Universal Robots PolyScope program: Calibration_6001.urp

Program Calibration_6001 (installation=GD directory=/programs/GD createdIn=5.13.0 lastSavedIn=5.13.0 robotSerialNumber=20205000017)
Calibrated DH parameters: a=[-0.000157, -0.56303, -0.236706, -0.000074, -0.000109, 0]; d=[0.181705, 47.632387, 369.599619, -417.058513, 0.119878, 0.115667]; alpha=[1.570881, -0.005074, -0.001247, 1.56886, -1.570997, 0]; deltaTheta=[0, -0.405485, 5.544791, 1.143886, -0.000009, -0.000001]
InitVariablesNode
BeforeStart
  Script file /programs/GD/ROVI/ROVI_RESET.script
    | def ROVI_RESET():
    |   if (not socket_open(host,port,socket_name)):
    |     rovi_err=902
    |     return False
    |   end
    |   socket_send_line("X0()",socket_name)
    |   ret=socket_read_line(socket_name,socket_timeout)
    |   if (ret == "OK"):
    |     rovi_err=0
    |   elif (ret == "NG"):
    |     rovi_err=to_num(socket_read_line(socket_name,socket_timeout))
    |   else:
    |     ret="NG"
    |     rovi_err=903
    |   end
    |   socket_close(socket_name)
    |   if (rovi_err != 0):
    |     if (is_popup):
    |       popup(str_cat(ret,rovi_err),title="X0",warning=True,blocking=True)
    |     end
    |     return False
    |   else:
    |     return True
    |   end
    | end
  Script file /programs/GD/ROVI/ROVI_CAPTURE.script
    | def ROVI_CAPTURE():
    | #  p=get_actual_tool_flange_pose()
    |   p=Bucket
    |   if (not socket_open(host,port,socket_name)):
    |     rovi_err=902
    |     return False
    |   end
    |   socket_send_string("X1(",socket_name)
    |   socket_send_string(p[0],socket_name)
    |   socket_send_string(",",socket_name)
    |   socket_send_string(p[1],socket_name)
    |   socket_send_string(",",socket_name)
    |   socket_send_string(p[2],socket_name)
    |   socket_send_string(",",socket_name)
    |   socket_send_string(p[3],socket_name)
    |   socket_send_string(",",socket_name)
    |   socket_send_string(p[4],socket_name)
    |   socket_send_string(",",socket_name)
    |   socket_send_string(p[5],socket_name)
    |   socket_send_line(")",socket_name)
    |   ret=socket_read_line(socket_name,socket_timeout)
    |   if (ret == "OK"):
    |     rovi_err=0
    |     f=socket_read_ascii_float(4,socket_name,socket_timeout)
    |     while (f[0]!=4):
    |       sleep(0.3)
    |       f=socket_read_ascii_float(4,socket_name,socket_timeout)
    |     end
    |     i=0
    |     while (i<4):
    |       Y1[i]=f[i+1]
    |       i=i+1
    |     end
    |   elif (ret == "NG"):
    |     rovi_err=to_num(socket_read_line(socket_name,socket_timeout))
    |   else:
    |     ret="NG"
    |     rovi_err=903
    |   end
    |   socket_close(socket_name)
    |   if (rovi_err != 0):
    |     if (is_popup):
    |       popup(str_cat(ret,rovi_err),title="X1",warning=True,blocking=True)
    |     end
    |     return False
    |   else:
    |     return True
    |   end
    | end
  Script file /programs/GD/ROVI/ROVI_SOLVE.script
    | def ROVI_SOLVE(is_popup=is_popup):
    |   buf=p[10000.0,0.0,0.0,0.0,0.0,0.0]
    |   if (not socket_open(host,port,socket_name)):
    |     rovi_err=902
    |     return False
    |   end
    |   socket_send_line("X2()",socket_name)
    |   ret=socket_read_line(socket_name,socket_timeout)
    |   if (ret == "OK"):
    |     rovi_err=0
    |     f=socket_read_ascii_float(6,socket_name,socket_timeout)
    |     while (f[0]!=6):
    |       sleep(0.3)
    |       f=socket_read_ascii_float(6,socket_name,socket_timeout)
    |     end
    |     counter=0
    |     while (counter<6):
    |       buf[counter]=f[counter+1]
    |       counter=counter+1
    |     end
    |   elif (ret == "NG"):
    |     rovi_err=to_num(socket_read_line(socket_name,socket_timeout))
    |   else:
    |     ret="NG"
    |     rovi_err=903
    |   end
    |   sleep(1.0)
    |   socket_close(socket_name)
    |   if (rovi_err != 0):
    |     if (is_popup):
    |       popup(str_cat(ret,rovi_err),title="X2",warning=True,blocking=True)
    |     end
    |   end
    |   return buf
    | end
Robot Program (runOnlyOnce=true)
  Call SUB_001
  Call SUB_6001
  Call SUB_001
SubProgram  [hidden by the author, left out]
SubProgram  [hidden by the author, left out]
SubProgram SUB_001 [hidden by the author, left out]
SubProgram SUB_6001 [hidden by the author, left out]
